FUNCTION_BLOCK EL3483
VAR
	_io : EL3483_Data;
	{attribute addProperty Name "WcState"}
	_wcState : WcStateInputToggle;
	{attribute addProperty Name "Info data"}
	_infoData : InfoDataAds;
END_VAR

PROPERTY IO : REFERENCE TO EL3483_Data
GET
IO REF= _io;
END_GET
END_PROPERTY

PROPERTY WcState : REFERENCE TO WcStateInputToggle
GET
WcState REF= _wcState;
END_GET
END_PROPERTY

END_FUNCTION_BLOCK

(* stored: Version 1.1.0.1, ProductVersion 3.1.4024.9
   POU EL3483: Id {bd8d4db1-6c35-05ec-3694-e2664d2b4036}, SpecialFunc None
   Property IO: Id {f130d515-1aca-0189-0a29-7348d77f85ad}
   Get Get: Id {7494767e-5b45-011b-15ef-8c76421cd251}
   Property WcState: Id {d448308a-654a-0c5e-1c54-ed10bb5be6be}
   Get Get: Id {aebc04c5-f074-0ea9-1eed-386bd9d43c50} *)
